(* IEC 61131-3 sources: 2026_Projet_YGO_ExcavatriceDragage/TOOLS/TEST_AUTO_CI/RESULTS/_TROUBLESHOOTING/t164_4c_encoder_compile, 5 files *)

(* ---- ST_EncoderMeasurement.st ---- *)
(* =======================================================================
   📊 ST_EncoderMeasurement — Mesures codeur conditionnées (1 sous-DUT par treuil)
   ───────────────────────────────────────────────────────────────
   🎯 Rôle : Regroupement des mesures et faits de la chaîne codeur d'un treuil (Abs → Scale → Safety → Speed)
   🔌 Interface : Interface de mesure normalisée pour PRG_02_Acquisition
   📄 Doc métier : DOC/AF/AF_Partie-06_Acquisition_Qualification_IO_v2.4.md
   ======================================================================= *)

TYPE ST_EncoderMeasurement :
STRUCT
    // === DONNEES BRUTES & STATUT BUS ===
    RawPos            : UDINT;        // Position brute codeur (gelee si EncoderAvailable=FALSE)
    EncoderAvailable  : BOOL;         // TRUE = bus/esclave EtherCAT operationnel et disponible

    // === MESURES DE POSITION CABLE ===
    CablePosM         : REAL;         // Position cable (m, signee, + enroule)
    CablePosMSafe     : REAL;         // Position cable instantanee validee par EncoderIncoherent (m)
    EncoderIncoherent : BOOL;         // TRUE = incoherence redemarrage ou hors bornes

    // === MESURES DE VITESSE CABLE ===
    Speed_Mps         : REAL;         // Vitesse absolue sur fenetre glissante (m/s)
    SignedSpeed_Mps   : REAL;         // Vitesse signee (m/s, + montee, - descente)
    SpeedValid        : BOOL;         // TRUE si 6 echantillons valides sur au moins 50 ms

    // === STATUTS DES SOUS-FB & REFERENCE ===
    HomingStatus      : ST_Status;  // Statut FB_Encoder_Homing (etat du referencement)
    AbsStatus         : ST_Status;  // Statut FB_Encoder_Abs (etat acquisition bus)
    HomingRefRaw      : UDINT;        // Reference brute du dernier homing reussi (re-expose)
END_STRUCT
END_TYPE

(* ---- FB_Encoder.st ---- *)
(* =======================================================================
   🔌 FB_Encoder — Objet codeur complet (1 par treuil M1/M2)
   ───────────────────────────────────────────────────────────────
   🎯 Rôle : Regrouper toute la chaine codeur derriere une interface unique :
      Abs → Homing → Scale → Safety → Reliability → Speed.
   🔌 Frontiere hardware separee HwIn/HwOut (testable).
   🔒 Homing : autorise par HomingPermit (calcule par le caller), declenche
      par HomingAtTargetM (front). La cible est fournie par le caller.
   🔒 Fiabilite : gate EncoderFault (sans Homed) calcule AVANT Speed — purge
      de vitesse au meme scan. HomedAndReliable = gate strict interlock M3.
   📄 Doc : DOC/AF/AF_Partie-09_Fonction_Encoder_v2.3.md
   ======================================================================= *)

FUNCTION_BLOCK FB_Encoder
VAR_INPUT
    // === COMMANDES & AUTORISATIONS ===
    Enable                : BOOL;        // --> [CMD] Autorisation generale FB (TRUE=Autorise)
    Reset                 : BOOL;        // --> [CMD] Acquittement defaut (front montant)

    // === AUTORISATION HOMING (calculee par le caller PRG) ===
    HomingPermit          : BOOL;        // --> [CMD] TRUE = l'operateur a le droit de homer

    // === CONSIGNES HOMING ===
    HomingAtTargetM       : BOOL;        // --> [CMD] Demande homing vers cible (front montant)
    HomingAtZero          : BOOL;        // --> [CMD] Force homing a 0.0
    ConfirmCoherence      : BOOL;        // --> [CMD] Lever le doute d'incoherence boot
    CfgHomingTargetM      : REAL;        // --> [CFG] Cible libre homing unitaire (m)
    CfgTopSensorPosM      : REAL;        // --> [CFG] Cible homing nominal capteur haut (m)
    UseDynamicTarget      : BOOL;        // --> [CMD] Active cible dynamique
    DynamicHomingTargetM  : REAL;       // --> [CFG] Cible dynamique de referencement (m)

    // === CAPTEURS PHYSIQUES ===
    TopPositionSensor     : BOOL;        // --> [HW]  Capteur physique position haute unique

    // === BUS ETHERCAT & CAPTEUR HW (frontiere testable) ===
    HwIn                  : ST_fbEncoder_HwIn; // --> [HW] Retours hardware codeur

    // === MECANIQUE (constantes) ===
    PointsPerRev          : UDINT := 8192; // --> [CFG] Resolution codeur (pts/tour)
    CableM_PerRev         : REAL := 2.0;   // --> [CFG] Developpement cable par tour (m/tour)

    // === REGLAGES & CONFIGURATION ===
    Cfg                   : ST_fbEncoder_Cfg; // --> [CFG] Mode de confirmation preset
    PositionMinM          : REAL := -99.0; // --> [CFG] Plafond bornage physique bas (m)
    PositionMaxM          : REAL := 99.0;  // --> [CFG] Plafond bornage physique haut (m)
    BypassGlobal          : BOOL := FALSE; // --> [TST] Neutralisation defauts pour mise en service
END_VAR
VAR_OUTPUT
    // === ETATS IEC & SYNOPTIQUE ===
    Ready                 : BOOL;        // <-- [STAT] FB pret a fonctionner
    Status                : ST_Status; // <-- [STAT] Statut transverse facade (synthese)

    // === FRONTIERE HW SORTIE (testable) ===
    HwOut                 : ST_fbEncoder_HwOut; // <-- [ACT] Ordres hardware codeur (preset)

    // === MESURES CONDITIONNEES (struct frontiere) ===
    Measurement           : ST_EncoderMeasurement; // <-- [BUS] Mesures + statuts (interface)

    // === ETATS CODEUR ===
    Homed                 : BOOL;        // <-- [STAT] Codeur reference (sortie homing)
    HomingSuspect         : BOOL;        // <-- [DIAG] Incoherence redemarrage a lever
    EncoderFault          : BOOL;        // <-- [SAFE] Gate general fiabilite (sans Homed)
    HomedAndReliable      : BOOL;        // <-- [STAT] Gate strict M3 : dispo ET ref ET pas incoherent
    PresetConfirmationFailed : BOOL;     // <-- [DIAG] Latch derniere verification preset echouee
END_VAR
VAR
    // === SOUS-INSTANCES FB (chaine codeur complete) ===
    instAbs        : FB_Encoder_Abs;          // * [INST] Acquisition brute codeur EtherCAT
    instHoming     : FB_Encoder_Homing;       // * [INST] Referencement (homing) nominal/unitaire
    instScale      : FB_Encoder_Scale;        // * [INST] Mise a l'echelle points -> metres
    instSafety     : FB_Encoder_Safety;       // * [INST] Bornage & coherence mesure
    instRel        : FB_EncoderReliability;   // * [INST] Gates de fiabilite
    instSpeed      : FB_Encoder_SpeedMeasure; // * [INST] Calcul vitesse cable
END_VAR
VAR_IN_OUT
    // === CALIBRATION PERSISTANTE (externe RETAIN, jamais membre) ===
    Calib                  : ST_Encoder_Calib; // <-> [BUS] Calibration RETAIN du treuil
END_VAR

IF NOT Enable THEN
    Ready := FALSE; Status.Busy := FALSE; Status.Done := FALSE; Status.Error := FALSE; Status.ErrorId := 16#0000;
    Status.State := E_State.DISABLED;
    Measurement.RawPos := 0; Measurement.EncoderAvailable := FALSE;
    Measurement.CablePosM := 0.0; Measurement.CablePosMSafe := 0.0; Measurement.EncoderIncoherent := FALSE;
    Measurement.Speed_Mps := 0.0; Measurement.SignedSpeed_Mps := 0.0; Measurement.SpeedValid := FALSE;
    Measurement.HomingStatus.State := E_State.DISABLED; Measurement.HomingStatus.Error := FALSE; Measurement.HomingStatus.ErrorId := 16#0000;
    Measurement.AbsStatus.State := E_State.DISABLED;    Measurement.AbsStatus.Error := FALSE;    Measurement.AbsStatus.ErrorId := 16#0000;
    EncoderFault := TRUE;
    HomedAndReliable := FALSE;
    // Frontiere HW sortie : aucun ordre preset publie hors autorisation
    // (sinon PRG_02_Acquisition relaie une valeur perimee au codeur absolu -> preset parasite, reference corrompue)
    HwOut.PresetTriggerCmd := 0; HwOut.CodeSeqTriggerCmd := 0; HwOut.PresetValueOut := 0;
    // Reference connue MAINTENUE depuis Calib (RETAIN) meme FB desactive (AF09 §4) :
    // un FB desactive ne doit pas faire perdre la reference aux consommateurs aval (PRG_04, FB_Encoder_Scale).
    Homed := Calib.Homed;
    HomingSuspect := Calib.HomingSuspect;
    Measurement.HomingRefRaw := Calib.HomingRefRaw;
    // PresetConfirmationFailed est un diagnostic latch : il reste gele hors Enable
    // et ne doit pas etre efface par ce gate (AC3).
    RETURN;
END_IF;
Ready := TRUE;
Status.State := E_State.READY;

    instAbs(
    Enable              := Enable,
    Reset               := Reset,
    RawPosIn            := HwIn.RawPosIn,
    AlarmsIn            := HwIn.AlarmsIn,
    WarningsIn          := HwIn.WarningsIn,
    SlaveOperational    := HwIn.SlaveOperational,
    PresetRequest       := instHoming.PresetRequest,
    PresetValue         := instHoming.PresetValue,
    PointsPerRev        := PointsPerRev
);

instHoming(
    Enable               := Enable,
    Reset                := Reset,
    Home                 := HomingAtTargetM,
    HomingPermit         := HomingPermit,
    BtnConfirmCoherence  := ConfirmCoherence,
    UseDynamicTarget     := UseDynamicTarget,
    DynamicHomingTargetM := DynamicHomingTargetM,
    CfgHomingTargetM     := CfgHomingTargetM,
    CfgTopSensorPosM     := SEL(HomingAtZero, CfgTopSensorPosM, 0.0),
    TopPositionSensor    := TopPositionSensor,
    RawPos               := instAbs.RawPos,
    EncoderAvailable     := instAbs.EncoderAvailable,
    PresetStatusBit      := HwIn.PresetStatusBit,
    Cfg                  := Cfg,
    PointsPerRev         := PointsPerRev,
    MultiTurnRevsMax     := 4096,
    CableM_PerRev        := CableM_PerRev,
    BypassGlobal         := BypassGlobal,
    Calib                := Calib
);

instScale(
    RawPos       := instAbs.RawPos,
    HomingRefRaw := instHoming.HomingRefRaw,
    CableM_PerRev := CableM_PerRev,
    PointsPerRev := PointsPerRev
);

instSafety(
    Enable             := Enable,
    Reset              := Reset,
    CablePosM          := instScale.CablePosM,
    HomingSuspect      := instHoming.HomingSuspect,
    PositionMinM       := PositionMinM,
    PositionMaxM       := PositionMaxM,
    BypassGlobal       := BypassGlobal
);

instRel(
    EncoderAvailable  := instAbs.EncoderAvailable,
    Homed             := instHoming.Homed,
    EncoderIncoherent := instSafety.EncoderIncoherent
);

instSpeed(
    Enable        := Enable,
    Reset         := Reset,
    Position_M    := instSafety.CablePosMSafe,
    PositionValid := NOT instRel.EncoderFault
);

Measurement.RawPos            := instAbs.RawPos;
Measurement.EncoderAvailable  := instAbs.EncoderAvailable;
Measurement.CablePosM         := instSafety.CablePosMSafe;
Measurement.CablePosMSafe     := instSafety.CablePosMSafe;
Measurement.EncoderIncoherent := instSafety.EncoderIncoherent;
Measurement.Speed_Mps         := instSpeed.Speed_Mps;
Measurement.SignedSpeed_Mps   := instSpeed.SignedSpeed_Mps;
Measurement.SpeedValid        := instSpeed.Valid;
Measurement.HomingStatus      := instHoming.Status;
Measurement.AbsStatus         := instAbs.Status;
Measurement.HomingRefRaw      := instHoming.HomingRefRaw;

// Frontiere HW sortie (preset)
HwOut.PresetTriggerCmd := instAbs.PresetTriggerCmd;
HwOut.CodeSeqTriggerCmd := instAbs.CodeSeqTriggerCmd;
HwOut.PresetValueOut    := instAbs.PresetValueOut;

// Etats codeur
Homed            := instHoming.Homed;
HomingSuspect    := instHoming.HomingSuspect;
EncoderFault     := instRel.EncoderFault;
HomedAndReliable := instRel.HomedAndReliable;
PresetConfirmationFailed := instHoming.PresetConfirmationFailed;

// Synthese statut facade
Status.Busy := instAbs.Status.Busy;
Status.Done := instSpeed.Valid AND instAbs.Ready;
Status.Error := instAbs.Status.Error OR instSafety.Status.Error OR instHoming.Status.Error;
Status.ErrorId := instAbs.Status.ErrorId OR instSafety.Status.ErrorId OR instHoming.Status.ErrorId;
END_FUNCTION_BLOCK

(* ---- FB_Encoder_Abs.st ---- *)
(* =======================================================================
   🔌 FB_Encoder_Abs — Acquisition codeur absolu (accès bus EtherCAT)
   ───────────────────────────────────────────────────────────────
   🎯 Rôle : Accès bus EtherCAT, extraction positions brutes et séquence de Preset SDO
   🔒 Polarité : EncoderAvailable=TRUE si communication bus et esclave OK
   🔌 Architecture : Module d'acquisition codeur absolu
   📄 Doc métier : DOC/AF/AF_Partie-09_Fonction_Encoder_v2.3.md
   ======================================================================= *)

// === DECLARATION (à coller dans la partie déclaration du POU FB_Encoder_Abs) ===

FUNCTION_BLOCK FB_Encoder_Abs
VAR_INPUT
    // === COMMANDES & AUTORISATIONS ===
    Enable              : BOOL;        // --> [CMD] Autorisation generale FB (TRUE=Autorise)
    Reset               : BOOL;        // --> [CMD] Acquittement defaut (front montant)
    PresetRequest       : BOOL;        // --> [CMD] Demande de preset (front montant)

    // === BUS ETHERCAT & CAPTEUR HW ===
    RawPosIn            : UDINT;       // --> [HW]  Position brute EtherCAT
    AlarmsIn            : UINT;        // --> [HW]  Codes alarmes bruts EtherCAT
    WarningsIn          : UINT;        // --> [HW]  Codes avertissements bruts EtherCAT
    SlaveOperational    : BOOL;        // --> [HW]  Statut esclave EtherCAT operationnel

    // === PARAMETRES & REGLAGES ===
    PointsPerRev        : UDINT := 8192; // --> [CFG] Resolution codeur (pts/tour)
    PresetValue         : UDINT;       // --> [CFG] Valeur cible de preset
    PresetTimeout       : TIME := T#2s;// --> [CFG] Temporisation max attente preset
    PresetTolerancePts  : UDINT := 10; // --> [CFG] Tolerance relecture post-preset (pts)
END_VAR
VAR_OUTPUT
    // === ETATS IEC & SYNOPTIQUE ===
    Ready               : BOOL;        // <-- [STAT] FB pret a fonctionner
    // 🧩 Statut transverse (forme cible) — regroupe Busy/Done/Error/ErrorId/State/StateAtError.
    // ErrorId bit0: "Com", bit1: "Preset Timeout".
    Status              : ST_Status;

    // === MESURES & DONNEES CODEUR ===
    RawPos              : UDINT;       // <-- [DIAG] Position brute gelee si non disponible
    EncoderAvailable    : BOOL;        // <-- [STAT] Codeur operationnel et disponible
    AngleRaw            : UINT;        // <-- [DIAG] Angle brut sur un tour (MOD PointsPerRev)
    TurnCount           : UDINT;       // <-- [DIAG] Nombre de tours bruts (RawPos / PointsPerRev)

    // === COMMANDES & ECHANGE BUS ETHERCAT ===
    PresetTriggerCmd    : WORD;        // <-- [ACT]  Ordre declenchement preset vers PDO Rx
    CodeSeqTriggerCmd   : WORD;        // <-- [ACT]  Ordre sequence code vers PDO Rx
    PresetValueOut      : UDINT;       // <-- [ACT]  Valeur de preset transmise au PDO Rx
END_VAR
VAR
    // === DETECTEURS DE FRONT ===
    ResetEdge           : R_TRIG;      // . [LOC] Detecteur front montant Reset
    ErrorEdge           : R_TRIG;      // . [LOC] Detecteur front montant Error
    PresetReqEdge       : R_TRIG;      // . [LOC] Detecteur front montant PresetRequest

    // === TEMPORISATEURS INTERNES ===
    PresetTimer         : TON;         // . [LOC] Temporisateur timeout sequence preset
    PresetTimerVisual   : TON;         // . [LOC] Temporisateur maintien visuel impulsion (500ms)

    // === VARIABLES INTERNES DE CALCUL & ETAT ===
    PresetSeqStep       : INT;         // . [LOC] Etape sequence preset (0:IDLE, 1:PULSE/WAIT)
    RawDiff             : DINT;        // . [LOC] Ecart signe entre RawPos et PresetValueOut
    PresetCompleted     : BOOL;        // . [LOC] Fait de fin de maintien preset (un scan)
END_VAR

// === IMPLEMENTATION (à coller dans le corps ST du POU FB_Encoder_Abs) ===

// 🛑 1. GATE
IF NOT Enable THEN
    EncoderAvailable := FALSE;
    Status.State := E_State.DISABLED;
    Ready := FALSE; Status.Busy := FALSE; Status.Done := FALSE;
    PresetTriggerCmd := 16#0000; CodeSeqTriggerCmd := 16#0000; PresetValueOut := 0;
    PresetSeqStep := 0;
    PresetCompleted := FALSE;
    PresetTimer(IN := FALSE, PT := PresetTimeout);
    PresetTimerVisual(IN := FALSE, PT := T#500MS);
    // RawPos, AngleRaw et TurnCount sont volontairement gelés hors Enable
    // (AF09 F09.01 / AC5) : aucune lecture bus ni remise a zero dans ce gate.
    RETURN;
END_IF;

Ready := TRUE;
Status.State := E_State.READY;

// 🔑 2. RESET FRONT
ResetEdge(CLK := Reset);

// 🔍 3. DIAGNOSTIC BUS / ALARME
IF (AlarmsIn <> 0) OR NOT SlaveOperational THEN
    Status.ErrorId := Status.ErrorId OR 16#0001;
ELSE
    Status.ErrorId := Status.ErrorId AND 16#FFFE; (* Auto-clearing dès que le bus et l'esclave sont OK *)
END_IF;
EncoderAvailable := (Status.ErrorId AND 16#0001) = 0;

// 📥 4. LECTURE POSITION — GELER SUR DOUTE (Partie10 §6)
// Si EncoderAvailable=FALSE : RawPos/AngleRaw/TurnCount conservent leur dernière valeur (pas de RETURN
// global ici pour ne pas geler aussi la séquence preset/l'état — seule la lecture est gelée).
IF EncoderAvailable THEN
    RawPos := RawPosIn;   // Sens de comptage géré côté codeur (CoE 6000h bit0, startup parameter CODESYS) — voir Partie10 §3bis. Plus de calcul ici.
    AngleRaw := UDINT_TO_UINT(RawPos MOD PointsPerRev);
    TurnCount := RawPos / PointsPerRev;
END_IF;

// 🔧 5. SÉQUENCE PRESET (écriture bus)
// PresetTriggerCmd := 2 déclenche le référencement à PresetValue (valeur de commande, pas un
// masque de bits). CodeSeqTriggerCmd : rôle non identifié — laissé à 0, PAS piloté tant que sa
// fonction n'est pas confirmée. Ne jamais lui donner une valeur arbitraire.
PresetReqEdge(CLK := PresetRequest);
PresetCompleted := FALSE;
CodeSeqTriggerCmd := 16#0000;           // non piloté — rôle inconnu, voir note ci-dessus
CASE PresetSeqStep OF
    0: // IDLE
        PresetTriggerCmd := 0;
        IF PresetReqEdge.Q AND EncoderAvailable THEN
            PresetValueOut := PresetValue;
            PresetSeqStep := 1;
            PresetTimer(IN := TRUE, PT := PresetTimeout);
        END_IF;
    1: // Déclenchement preset (laissé actif pendant 0.5s pour confort visuel en simulation/bus)
        PresetTriggerCmd := 2;   // Référence le codeur à PresetValueOut
        RawDiff := UDINT_TO_DINT(RawPos) - UDINT_TO_DINT(PresetValueOut);
        IF ABS(RawDiff) <= UDINT_TO_DINT(PresetTolerancePts) THEN
            PresetTimer(IN := FALSE, PT := PresetTimeout);
            PresetTimerVisual(IN := TRUE, PT := T#500MS);
            IF PresetTimerVisual.Q THEN
                PresetTriggerCmd := 0;
                PresetCompleted := TRUE;
                PresetSeqStep := 0;
                PresetTimerVisual(IN := FALSE, PT := T#500MS);
            END_IF;
        ELSIF PresetTimer.Q THEN
            PresetTriggerCmd := 0;
            Status.ErrorId := Status.ErrorId OR 16#0002;
            PresetSeqStep := 0;
            PresetTimer(IN := FALSE, PT := PresetTimeout);
            PresetTimerVisual(IN := FALSE, PT := T#500MS);
        END_IF;
END_CASE;
IF ResetEdge.Q AND (PresetSeqStep = 0) THEN
    Status.ErrorId := Status.ErrorId AND 16#FFFD;
END_IF;

// 🧾 6. ERROR / STATEATERROR
Status.Error := (Status.ErrorId <> 16#0000);
ErrorEdge(CLK := Status.Error);
IF ErrorEdge.Q THEN
    Status.StateAtError := Status.State;
END_IF;

Status.Busy := (PresetSeqStep <> 0);
Status.Done := PresetCompleted;
END_FUNCTION_BLOCK

(* ---- FB_Encoder_Homing.st ---- *)
(* =======================================================================
   ⚙️ FB_Encoder_Homing — Référencement codeur nominal ou unitaire
   ───────────────────────────────────────────────────────────────
   🎯 Rôle : Séquence de référencement nominal (capteur haut) ou unitaire (MAINT_N2)
   🔒 Polarité : Homed=TRUE dès qu'un référencement valide est enregistré
   🔌 Architecture : Expose ST_Encoder_Calib en VAR_IN_OUT
   📄 Doc métier : DOC/AF/AF_Partie-09_Fonction_Encoder_v2.3.md
   ======================================================================= *)

// === DECLARATION (à coller dans la partie déclaration du POU FB_Encoder_Homing) ===

FUNCTION_BLOCK FB_Encoder_Homing
VAR_INPUT
    // === COMMANDES & AUTORISATIONS ===
    Enable                 : BOOL;        // --> [CMD] Autorisation generale FB (TRUE=Autorise)
    Reset                  : BOOL;        // --> [CMD] Acquittement defaut (front montant)
    Home                   : BOOL;        // --> [CMD] Demande de referencement (front)
    HomingPermit           : BOOL;        // --> [CMD] Autorisation de homer (calculee par le caller)
    BtnConfirmCoherence    : BOOL;        // --> [CMD] Levee de doute d'incoherence au boot (front)

    // === CIBLES & CONFIGURATION HOMING ===
    CfgHomingTargetM       : REAL;        // --> [CFG] Cible libre homing unitaire (m)
    UseDynamicTarget       : BOOL := FALSE; // --> [CFG] Activation cible dynamique
    DynamicHomingTargetM   : REAL := 0.0; // --> [CFG] Cible dynamique de referencement (m)
    CfgTopSensorPosM       : REAL := 8.5; // --> [CFG] Cible homing nominal capteur haut (m)

    // === RETOURS HW & CAPTEURS ===
    TopPositionSensor      : BOOL;        // --> [HW]  Capteur physique position haute unique
    // === MESURES & RETOURS FB CODEUR ABSOLU ===
    RawPos                 : UDINT;       // --> [HW]  Position brute codeur (sortie FB_Encoder_Abs)
    EncoderAvailable       : BOOL;        // --> [HW]  Codeur absolu disponible et valide
    PresetStatusBit        : BOOL;        // --> [HW]  Bit d'etat preset optionnel, FALSE si non cable

    // === REGLAGES TRANSACTION PRESET ===
    Cfg                    : ST_fbEncoder_Cfg; // --> [CFG] Mode de confirmation preset

    // === CARACTERISTIQUES MECANIQUES & BUS ===
    PointsPerRev           : UDINT := 8192; // --> [CFG] Resolution codeur (pts/tour)
    MultiTurnRevsMax       : UDINT := 4096; // --> [CFG] Capacite multitour max codeur (tours)
    CableM_PerRev          : REAL := 2.0;   // --> [CFG] Perimetre tambour / developpement cable (m/tour)

    // === TESTS & BYPASS ===
    BypassGlobal           : BOOL := FALSE; // --> [TST] Neutralisation securites pour mise en service
END_VAR
VAR_OUTPUT
    // === ETATS IEC & SYNOPTIQUE ===
    Ready                  : BOOL;        // <-- [STAT] FB pret a fonctionner
    // 🧩 Statut transverse (forme cible) — regroupe Busy/Done/Error/ErrorId/State/StateAtError.
    // ErrorId : masque de bits de défaut (bit0: mode, bit1: treuil, bit4: cible, bit5: preset, bit9: incoherence boot).
    Status                 : ST_Status;

    // === COMMANDES VERS FB_ENCODER_ABS ===
    PresetRequest          : BOOL;        // <-- [ACT]  Pulse demande d'ecriture preset SDO
    PresetValue            : UDINT;       // <-- [ACT]  Valeur de cible brute pour preset SDO

    // === RESULTATS & MEMOIRE CALIBRATION ===
    Homed                  : BOOL;        // <-- [STAT] Codeur pagine et referencie
    HomingSuspect          : BOOL;        // <-- [DIAG] Incoherence redemarrage a lever
    HomingRefRaw           : UDINT;       // <-- [DIAG] Offset de reference brut calcule
    PresetConfirmationFailed : BOOL;      // <-- [DIAG] Latch derniere verification preset echouee
END_VAR
VAR_IN_OUT
    // === STRUCTURE DE CALIBRATION PERSISTANTE ===
    Calib                  : ST_Encoder_Calib; // <-> [BUS] Structure de calibration RETAIN
END_VAR
VAR
    // === DETECTEURS DE FRONT ===
    ResetEdge              : R_TRIG;      // . [LOC] Detecteur front montant Reset
    ErrorEdge              : R_TRIG;      // . [LOC] Detecteur front montant Error
    HomeEdge               : R_TRIG;      // . [LOC] Detecteur front montant Home
    ConfirmCoherenceEdge   : R_TRIG;      // . [LOC] Detecteur front montant BtnConfirmCoherence
    TopSensorEdge          : R_TRIG;      // . [LOC] Detecteur front montant TopPositionSensor
    DynamicTargetEdge      : R_TRIG;      // . [LOC] Detecteur front montant UseDynamicTarget

    // === ETATS & DRAPEAUX INTERNES ===
    InitDone               : BOOL;        // . [LOC] Controle incoherence boot effectue
    ArretConfirme          : BOOL;        // . [LOC] Condition d'arret moteur confirmee
    HomingModeOk           : BOOL;        // . [LOC] Mode de fonctionnement valide pour homing
    NominalHomingTrigger   : BOOL;        // . [LOC] Condition de declenchement homing nominal
    UnitaryHomingTrigger   : BOOL;        // . [LOC] Condition de declenchement homing unitaire
    DynamicHomingTrigger   : BOOL;        // . [LOC] Condition de declenchement homing dynamique
    HomingTrigger          : BOOL;        // . [LOC] Synthese declenchement homing
    PresetVerificationActive : BOOL;      // . [LOC] Verification preset en attente
    PresetConfirmed        : BOOL;        // . [LOC] Resultat du mode de confirmation selectionne

    // === VARIABLES DE CALCUL ===
    TargetPoints           : DINT;        // . [LOC] Ecart cible converti en points
    TargetPositionM        : REAL;        // . [LOC] Cible retenue en metres
    RawDiffRestart         : DINT;        // . [LOC] Ecart brut de position au redemarrage
    PendingHomingRefRaw    : UDINT;       // . [LOC] Reference candidate, non publiee avant succes
    CandidateRawDiff       : DINT;        // . [LOC] Ecart brut de la mesure candidate
    CandidateCablePosM     : REAL;        // . [LOC] Position candidate calculee avant commit
    ReadbackOk             : BOOL;        // . [LOC] Mesure candidate dans la tolerance
    StatusBitOk             : BOOL;       // . [LOC] Etat du bit optionnel de confirmation
    PresetVerifyTimer       : TON;        // . [LOC] Temporisation historique de verification 500ms
END_VAR

VAR CONSTANT
    // === TOLERANCE & TEMPORISATION TRANSACTION ===
    CST_HomingVerifyToleranceM : REAL := 0.010; // Tolerance mesure cible (m)
    CST_PresetVerifyTime        : TIME := T#500MS; // Latence historique avant relecture
END_VAR

// === IMPLEMENTATION (à coller dans le corps ST du POU FB_Encoder_Homing) ===

// 🛑 1. GATE — neutralisation ; on continue toutefois d'exposer le dernier état RETAIN connu
// (FB_Encoder_Scale a besoin de HomingRefRaw même si ce FB est désactivé)
// PowerContactorEngaged retiré du GATE (le codeur 24V / EtherCAT peut être homé disjoncteurs coupés)
IF NOT Enable THEN
    PresetRequest := FALSE;
    PresetValue := 0;
    Status.State := E_State.DISABLED;
    Ready := FALSE; Status.Busy := FALSE; Status.Done := FALSE;
    InitDone := FALSE;   // Force un nouveau contrôle §3.7 à la prochaine activation
    PresetVerificationActive := FALSE;
    PresetVerifyTimer(IN := FALSE, PT := CST_PresetVerifyTime);
    Homed := Calib.Homed;
    HomingSuspect := Calib.HomingSuspect;
    HomingRefRaw := Calib.HomingRefRaw;
    // PresetConfirmationFailed est un diagnostic latch : il est gele hors Enable
    // et n'est ni valide ni efface par la desactivation (AC3).
    RETURN;
END_IF;

Ready := TRUE;

// 🔑 2. FRONTS
ResetEdge(CLK := Reset);
HomeEdge(CLK := Home);
ConfirmCoherenceEdge(CLK := BtnConfirmCoherence);

// 🔍 3. COHÉRENCE AU REDÉMARRAGE (§3.7) — une fois par session Enable, dès que le codeur répond
IF NOT InitDone THEN
    Status.State := E_State.INIT;
    IF EncoderAvailable THEN
        RawDiffRestart := UDINT_TO_DINT(RawPos) - UDINT_TO_DINT(Calib.LastKnownRawPos);
        IF Calib.Homed AND (ABS(RawDiffRestart) > UDINT_TO_DINT(Calib.RestartCoherenceTolerancePts)) THEN
            Calib.HomingSuspect := TRUE;
            Status.ErrorId := Status.ErrorId OR 16#0200;   // bit9 : incohérence codeur au redémarrage
        END_IF;
        InitDone := TRUE;
    END_IF;
ELSE
    IF Status.State = E_State.INIT THEN Status.State := E_State.READY; END_IF;
END_IF;

// ✅ 4. LEVÉE DU DOUTE (BtnConfirmCoherence, §3.7) — indépendant du Reset générique
IF ConfirmCoherenceEdge.Q AND HomingPermit THEN
    Calib.HomingSuspect := FALSE;
    Status.ErrorId := Status.ErrorId AND 16#FDFF;   // efface bit9
END_IF;

PresetRequest := FALSE;
PresetValue := 0;
TopSensorEdge(CLK := TopPositionSensor);
DynamicTargetEdge(CLK := UseDynamicTarget);

// Gates rejetées = Warning auto-effaçable (§9/TC-P03-007), pas un Fault : recalculées à
// chaque scan, jamais latchées, aucun Reset requis pour les effacer.
Status.ErrorId := Status.ErrorId AND 16#FFEC;   // efface bits 0/1/4 (garde bit5, bit9 — inchangés)

HomingModeOk := HomingPermit;

IF HomeEdge.Q AND NOT HomingModeOk THEN
    Status.ErrorId := Status.ErrorId OR 16#0001;   // bit0 : homing non autorise
END_IF;

// Nominal : capture AU FRONT du capteur haut, pas après arrêt confirmé — AscentPermit
// (FB_Safety_Winch) coupe déjà la montée indépendamment dès que TopPositionSensor est actif ;
// attendre l'arrêt casserait la répétabilité recherchée à vitesse d'accostage constante.
// Couvre les deux cas : Home déjà maintenu quand le capteur déclenche, ou capteur déjà actif
// quand Home est pressé.
NominalHomingTrigger := HomingModeOk AND NOT UseDynamicTarget
                         AND ((Home AND TopSensorEdge.Q) OR (HomeEdge.Q AND TopPositionSensor));

// Unitaire : cible libre (CfgHomingTargetM), déclenchée par la demande (front).
UnitaryHomingTrigger := HomingModeOk AND NOT UseDynamicTarget AND HomeEdge.Q;

// Dynamique (benne) : HomingModeOk vérifié ici en défense.
DynamicHomingTrigger := HomingModeOk AND (DynamicTargetEdge.Q OR (UseDynamicTarget AND HomeEdge.Q));

HomingTrigger := (NominalHomingTrigger OR UnitaryHomingTrigger OR DynamicHomingTrigger)
                 AND NOT PresetVerificationActive;

IF HomingTrigger THEN
    IF UseDynamicTarget THEN
        TargetPositionM := DynamicHomingTargetM;
    ELSIF NominalHomingTrigger THEN
        TargetPositionM := CfgTopSensorPosM;
    ELSE
        TargetPositionM := CfgHomingTargetM;
    END_IF;

    // Bornage obligatoire avant écriture (CODE_QUALITY_STANDARDS §6) — toute cible, quelle
    // que soit son origine (config, calcul benne, capteur haut), est vérifiée dans la plage
    // physique documentée [-99;+99] m avant d'être gravée dans la référence codeur.
    IF (TargetPositionM < -99.0) OR (TargetPositionM > 99.0) THEN
        Status.ErrorId := Status.ErrorId OR 16#0010;   // bit4 : cible hors plage, homing refusé
    ELSE
        TargetPoints := REAL_TO_DINT(TargetPositionM * UDINT_TO_REAL(PointsPerRev) / CableM_PerRev);
        PendingHomingRefRaw := DINT_TO_UDINT(UDINT_TO_DINT(RawPos) - TargetPoints);
        PresetValue := RawPos;
        PresetRequest := TRUE;
        PresetVerificationActive := TRUE;
        Status.Done := FALSE;
        // Le suivi transactionnel reste interne : ne pas publier BUSY, car ce
        // statut est consomme par PRG_04 comme mode de referencement securite.

        // Demande preset vers FB_Encoder_Abs ; la relecture mesuree est la seule
        // confirmation en READBACK_ONLY (mesure relue conforme a la cible).
    END_IF;
END_IF;

// ⏳ 6. SUIVI DE LA SÉQUENCE SDO OPTIONNELLE
PresetVerifyTimer(IN := PresetVerificationActive, PT := CST_PresetVerifyTime);
IF PresetVerificationActive AND PresetVerifyTimer.Q THEN
    CandidateRawDiff := UDINT_TO_DINT(RawPos) - UDINT_TO_DINT(PendingHomingRefRaw);
    IF PointsPerRev <> 0 THEN
        CandidateCablePosM := DINT_TO_REAL(CandidateRawDiff) * CableM_PerRev / UDINT_TO_REAL(PointsPerRev);
    ELSE
        CandidateCablePosM := 0.0;
    END_IF;
    ReadbackOk := ABS(CandidateCablePosM - TargetPositionM) <= CST_HomingVerifyToleranceM;
    StatusBitOk := PresetStatusBit;

    CASE Cfg.PresetConfirmMode OF
        E_PresetConfirmMode.READBACK_ONLY:
            PresetConfirmed := ReadbackOk;
        E_PresetConfirmMode.READBACK_AND_STATUSBIT:
            PresetConfirmed := ReadbackOk AND StatusBitOk;
        E_PresetConfirmMode.STATUSBIT_ONLY:
            PresetConfirmed := StatusBitOk;
        ELSE
            PresetConfirmed := FALSE;
    END_CASE;

    IF PresetConfirmed THEN
        Calib.HomingRefRaw := PendingHomingRefRaw;
        Calib.Homed := TRUE;
        Calib.HomingSuspect := FALSE;
        Calib.LastKnownRawPos := RawPos;
        PresetConfirmationFailed := FALSE;
        Status.ErrorId := Status.ErrorId AND 16#FFDF;
        Status.Done := TRUE;
    ELSE
        Calib.HomingSuspect := TRUE;
        PresetConfirmationFailed := TRUE;
        Status.ErrorId := Status.ErrorId OR 16#0020;
        Status.Done := FALSE;
    END_IF;

    PresetVerificationActive := FALSE;
    PresetVerifyTimer(IN := FALSE, PT := CST_PresetVerifyTime);
    Status.State := E_State.READY;
END_IF;

// 🧾 7. RESET (front) — efface les bits « dernière tentative rejetée » (pas de cause persistante
// à revérifier ici : le prochain Home réévalue toutes les conditions de zéro, voir §5)
IF ResetEdge.Q THEN
    PresetConfirmationFailed := FALSE;
    Status.ErrorId := Status.ErrorId AND 16#FFC0;   // efface bits 0..5 (garde bit9, levé seulement par BtnConfirmCoherence/Home)
END_IF;

// 📤 8. SORTIES ÉTAT
Status.Error := (Status.ErrorId <> 16#0000);
ErrorEdge(CLK := Status.Error);
IF ErrorEdge.Q THEN
    Status.StateAtError := Status.State;
END_IF;

// Mise à jour continue du point brut valide connu (hors séquence de homing elle-même)
IF EncoderAvailable AND (Status.State <> E_State.BUSY) THEN
    Calib.LastKnownRawPos := RawPos;
END_IF;

Status.Busy := (Status.State = E_State.BUSY);
Homed := Calib.Homed AND NOT Calib.HomingSuspect; // Perd l'état homed si suspect (démarrage ou fonctionnement), restauré après BtnConfirmCoherence
HomingSuspect := Calib.HomingSuspect;
HomingRefRaw := Calib.HomingRefRaw;
END_FUNCTION_BLOCK

(* ---- FB_Encoder_SpeedMeasure.st ---- *)
(* =======================================================================
   ⚙️ FB_Encoder_SpeedMeasure — Mesure de vitesse câble horodatée
   ───────────────────────────────────────────────────────────────
   🎯 Rôle : Calcul de la vitesse absolue et signée sur fenêtre glissante horodatée
   🔒 Polarité : Valid=TRUE après 6 échantillons couvrant au moins 50ms
   📄 Doc métier : DOC/AF/AF_Partie-09_Fonction_Encoder_v2.3.md
   ======================================================================= *)

FUNCTION_BLOCK FB_Encoder_SpeedMeasure
VAR_INPUT
    // === COMMANDES & AUTORISATIONS ===
    Enable              : BOOL;        // --> [CMD] Autorisation generale FB (TRUE=Autorise)
    Reset               : BOOL;        // --> [CMD] Purge immediate de l'historique (front montant)

    // === MESURE SURES EN ENTREE ===
    Position_M          : REAL;        // --> [HW]  Position cable sure en metres (FB_Encoder_Safety)
    PositionValid       : BOOL;        // --> [SAFE] Validite de la chaine codeur
END_VAR
VAR_OUTPUT
    // === VITESSE CALCULÉE & VALIDITE ===
    Speed_Mps           : REAL;        // <-- [DIAG] Vitesse absolue sur la fenetre glissante (m/s)
    SignedSpeed_Mps     : REAL;        // <-- [DIAG] Vitesse signee (+ montee, - descente) (m/s)
    Valid               : BOOL;        // <-- [STAT] Vitesse valide (6 ech. sur 50 ms)
END_VAR
VAR
    // === HISTORIQUE & ECHANTILLONS ===
    Positions_M         : ARRAY[0..5] OF REAL; // . [LOC] Tableau des 6 positions enregistrees
    Timestamps          : ARRAY[0..5] OF TIME; // . [LOC] Horodatage associe aux 6 positions

    // === HORODATAGE & TEMPORISATION ===
    CurrentTimestamp    : TIME;        // . [LOC] Horodatage courant du cycle
    LastTimestamp       : TIME;        // . [LOC] Horodatage de l'echantillon precedent
    ElapsedSinceSample  : TIME;        // . [LOC] Temps ecoule depuis le dernier echantillon
    WindowElapsed       : TIME;        // . [LOC] Temps total ecoule sur la fenetre de mesure

    // === COMPTEURS & ETATS INTERNES ===
    CollectedSamples    : INT;         // . [LOC] Nombre d'echantillons collectes dans la fenetre
    Index               : INT;         // . [LOC] Index de boucle de decalage
    TimestampInitialized: BOOL;        // . [LOC] Indicateur d'initialisation du premier horodatage
END_VAR
VAR CONSTANT
    // === PARAMETRES DE LA FENETRE GLISSANTE ===
    WindowTime          : TIME := T#50MS; // Fenetre glissante de mesure
    SamplePeriod        : TIME := T#10MS; // Periode minimale entre deux echantillons
    SampleCount         : INT := 6;       // Nombre total d'echantillons requis
END_VAR

// ⏱️ Horodatage natif : le calcul utilise le temps réellement écoulé, jamais un cycle supposé.
CurrentTimestamp := TIME();

// Purge des six positions sur rupture de confiance : aucune source antérieure ne peut contaminer la mesure.
IF NOT Enable OR Reset OR NOT PositionValid THEN
    Speed_Mps := 0.0;
    SignedSpeed_Mps := 0.0;
    Valid := FALSE;
    CollectedSamples := 0;
    TimestampInitialized := FALSE;
    RETURN;
END_IF;

// 🕒 Première position de la nouvelle fenêtre.
IF NOT TimestampInitialized THEN
    Positions_M[0] := Position_M;
    Timestamps[0] := CurrentTimestamp;
    LastTimestamp := CurrentTimestamp;
    CollectedSamples := 1;
    TimestampInitialized := TRUE;
    Speed_Mps := 0.0;
    SignedSpeed_Mps := 0.0;
    Valid := FALSE;
    RETURN;
END_IF;

// 🛡️ Rebouclage de TIME détecté localement : purge sans réutiliser le delta aberrant.
IF CurrentTimestamp < LastTimestamp THEN
    Positions_M[0] := Position_M;
    Timestamps[0] := CurrentTimestamp;
    LastTimestamp := CurrentTimestamp;
    CollectedSamples := 1;
    Speed_Mps := 0.0;
    SignedSpeed_Mps := 0.0;
    Valid := FALSE;
    RETURN;
END_IF;

ElapsedSinceSample := CurrentTimestamp - LastTimestamp;

// 🛡️ Delta nul : aucune division et aucun doublon d'échantillon.
IF ElapsedSinceSample <= T#0MS THEN
    RETURN;
END_IF;

// 📥 Six positions espacées d'au moins 10 ms donnent cinq intervalles sur la fenêtre interne de 50 ms.
IF ElapsedSinceSample >= SamplePeriod THEN
    LastTimestamp := CurrentTimestamp;

    IF CollectedSamples < SampleCount THEN
        Positions_M[CollectedSamples] := Position_M;
        Timestamps[CollectedSamples] := CurrentTimestamp;
        CollectedSamples := CollectedSamples + 1;
    ELSE
        FOR Index := 0 TO 4 DO
            Positions_M[Index] := Positions_M[Index + 1];
            Timestamps[Index] := Timestamps[Index + 1];
        END_FOR;
        Positions_M[5] := Position_M;
        Timestamps[5] := CurrentTimestamp;
    END_IF;

    IF CollectedSamples = SampleCount THEN
        // 🛡️ Ordre temporel et durée minimale contrôlés avant toute conversion/division.
        IF Timestamps[5] >= Timestamps[0] THEN
            WindowElapsed := Timestamps[5] - Timestamps[0];
            IF WindowElapsed >= WindowTime THEN
                SignedSpeed_Mps := (Positions_M[5] - Positions_M[0])
                                   / (UDINT_TO_REAL(TIME_TO_UDINT(WindowElapsed)) / 1000.0);
                Speed_Mps := ABS(SignedSpeed_Mps);
                Valid := TRUE;
            ELSE
                Speed_Mps := 0.0;
                SignedSpeed_Mps := 0.0;
                Valid := FALSE;
            END_IF;
        ELSE
            Speed_Mps := 0.0;
            SignedSpeed_Mps := 0.0;
            Valid := FALSE;
            CollectedSamples := 0;
            TimestampInitialized := FALSE;
        END_IF;
    END_IF;
END_IF;
END_FUNCTION_BLOCK
